TYPE ST_ErgoCommands :
STRUCT
	Done : BOOL := FALSE;
END_STRUCT
END_TYPE

(* stored: Version 1.1.0.1, ProductVersion 3.1.4024.12
   DUT ST_ErgoCommands: Id {83e2c9a0-4a8e-48a3-99b4-9d0f36b7529f} *)
